(* CoDeSys 2.3 export: SENSORBATH.EXP *)

(* Data type in BathFB *)
TYPE SensorBath :
STRUCT
    level:			LevelBath;   (*Уровни*)
    tempBath:		REAL;        (*Температура ванны*)
    tempTank:		REAL;        (*Температура бака*)
	tempAir:		REAL;
	button:			ButtonBath;  (*Кнопки*)
    Fl:				FlE;         (*тип жидкости в ванне*)
    warmOn:			BOOL;        (*нагрев включен*)
    mixOn:			BOOL;        (*перемешивание включен*)
    pause:			BOOL;        (*Пауза АП*)
    rotOn:			BOOL;        (*Включение вращения*)
    flReset:		BOOL;        (*Сброс типа жидкости*)
	overloadPump:	BOOL;        (*перегрузка насоса*)
END_STRUCT
END_TYPE
